PROGRAM MAIN
VAR
	fbMover							: MC_PlanarMover;
	afbAxis							: ARRAY [1..6] OF AXIS_REF;
	fbXPlanarGamePad				: FB_XPlanarGamePad;
END_VAR

fbMover.Update();

fbXPlanarGamePad(
	fbMover:= fbMover, 
	fbMoverAxis:= afbAxis, 
	stGamePad:= GVL.stGamePad1, 
	lrStickDeadZone:= 3000, 
	stStatus=> );

END_PROGRAM

(* stored: Version 1.1.0.1
   POU MAIN: Id {3b2e30a5-fd08-4af5-bac7-164098d87b7b}, SpecialFunc None *)
